KUKA KRL program: scorepoints.src, scorepoints.dat

--- scorepoints.src ---
&ACCESS RVP
&REL 2
&PARAM EDITMASK = *
&PARAM TEMPLATE = C:\KRC\Roboter\Template\vorgabe
DEF scorepoints( )
;FOLD INI;%{PE}
  ;FOLD BASISTECH INI
    GLOBAL INTERRUPT DECL 3 WHEN $STOPMESS==TRUE DO IR_STOPM ( )
    INTERRUPT ON 3
    BAS (#INITMOV,0 )
  ;ENDFOLD (BASISTECH INI)
  ;FOLD USER INI
    ;Make your modifications here

  ;ENDFOLD (USER INI)
;ENDFOLD (INI)

;FOLD PTP HOME  Vel= 100 % DEFAULT;%{PE}%MKUKATPBASIS,%CMOVE,%VPTP,%P 1:PTP, 2:HOME, 3:, 5:100, 7:DEFAULT
$BWDSTART = FALSE
PDAT_ACT=PDEFAULT
FDAT_ACT=FHOME
BAS (#PTP_PARAMS,100 )
$H_POS=XHOME
PTP  XHOME
;ENDFOLD

;FOLD SLIN P1 Vel=2 m/s CPDAT1 Tool[15]:R2_educate_pro_MARKER Base[5]:paper;%{PE}%R 8.3.44,%MKUKATPBASIS,%CSPLINE,%VSLIN_SB,%P 1:SLIN_SB, 2:P1, 3:, 5:2, 7:CPDAT1
SLIN XP1 WITH $VEL=SVEL_CP( 2, , LCPDAT1), $TOOL=STOOL2( FP1), $BASE= SBASE( FP1.BASE_NO),$IPO_MODE=SIPO_MODE( FP1.IPO_FRAME), $LOAD=SLOAD( FP1.TOOL_NO), $ACC=SACC_CP( LCPDAT1), $ORI_TYPE=SORI_TYP( LCPDAT1), $JERK=SJERK( LCPDAT1)
;ENDFOLD
;FOLD SLIN P2 Vel=2 m/s CPDAT2 Tool[15]:R2_educate_pro_MARKER Base[5]:paper;%{PE}%R 8.3.44,%MKUKATPBASIS,%CSPLINE,%VSLIN_SB,%P 1:SLIN_SB, 2:P2, 3:, 5:2, 7:CPDAT2
SLIN XP2 WITH $VEL=SVEL_CP( 2, , LCPDAT2), $TOOL=STOOL2( FP2), $BASE= SBASE( FP2.BASE_NO),$IPO_MODE=SIPO_MODE( FP2.IPO_FRAME), $LOAD=SLOAD( FP2.TOOL_NO), $ACC=SACC_CP( LCPDAT2), $ORI_TYPE=SORI_TYP( LCPDAT2), $JERK=SJERK( LCPDAT2)
;ENDFOLD
;FOLD PTP HOME  Vel= 100 % DEFAULT;%{PE}%MKUKATPBASIS,%CMOVE,%VPTP,%P 1:PTP, 2:HOME, 3:, 5:100, 7:DEFAULT
$BWDSTART = FALSE
PDAT_ACT=PDEFAULT
FDAT_ACT=FHOME
BAS (#PTP_PARAMS,100 )
$H_POS=XHOME
PTP  XHOME
;ENDFOLD

END

--- scorepoints.dat ---
&ACCESS RVP
&REL 2
&PARAM EDITMASK = *
&PARAM TEMPLATE = C:\KRC\Roboter\Template\vorgabe
DEFDAT  scorepoints
;FOLD EXTERNAL DECLARATIONS;%{PE}%MKUKATPBASIS,%CEXT,%VCOMMON,%P
;FOLD BASISTECH EXT;%{PE}%MKUKATPBASIS,%CEXT,%VEXT,%P
EXT  BAS (BAS_COMMAND  :IN,REAL  :IN )
DECL INT SUCCESS
;ENDFOLD (BASISTECH EXT)
;FOLD USER EXT;%{E}%MKUKATPUSER,%CEXT,%VEXT,%P
;Make your modifications here

;ENDFOLD (USER EXT)
;ENDFOLD (EXTERNAL DECLARATIONS)
DECL BASIS_SUGG_T LAST_BASIS={POINT1[] "P2                      ",POINT2[] "P2                      ",CP_PARAMS[] "CPDAT2                  ",PTP_PARAMS[] "PDAT0                   ",CONT[] "                        ",CP_VEL[] "2                       ",PTP_VEL[] "100                     ",SYNC_PARAMS[] "SYNCDAT                 ",SPL_NAME[] "S0                      ",A_PARAMS[] "ADAT0                   "}
DECL E6POS XP1={X 520.892334,Y 120.634895,Z -44.3008270,A 111.070587,B 88.6128082,C -161.537918,S 2,T 35,E1 0.0,E2 0.0,E3 0.0,E4 0.0,E5 0.0,E6 0.0}
DECL FDAT FP1={TOOL_NO 15,BASE_NO 5,IPO_FRAME #BASE,POINT2[] " ",TQ_STATE FALSE}
DECL LDAT LCPDAT1={VEL 2.00000,ACC 100.000,APO_DIST 100.000,APO_FAC 50.0000,AXIS_VEL 100.000,AXIS_ACC 100.000,ORI_TYP #VAR,CIRC_TYP #BASE,JERK_FAC 50.0000,GEAR_JERK 50.0000,EXAX_IGN 0}
DECL E6POS XP2={X 571.230286,Y 120.628372,Z -44.4825401,A 111.078186,B 88.6129532,C -161.530258,S 2,T 35,E1 0.0,E2 0.0,E3 0.0,E4 0.0,E5 0.0,E6 0.0}
DECL FDAT FP2={TOOL_NO 15,BASE_NO 5,IPO_FRAME #BASE,POINT2[] " ",TQ_STATE FALSE}
DECL LDAT LCPDAT2={VEL 2.00000,ACC 100.000,APO_DIST 100.000,APO_FAC 50.0000,AXIS_VEL 100.000,AXIS_ACC 100.000,ORI_TYP #VAR,CIRC_TYP #BASE,JERK_FAC 50.0000,GEAR_JERK 50.0000,EXAX_IGN 0}
ENDDAT
